(* Schneider Machine Expert - Basic project Modelo final v0.4, file version 2.6.0.0 *)
(* ProjectInformations: Name=Nuevo proyecto *)

HARDWARE
  Cpu 0: TM221CE24T
  EthernetConfiguration: NetworkName=M221, IpAllocationMode=FixedAddress, IpAddress=0.0.0.0, SubnetMask=0.0.0.0
  SerialLineConfiguration: Baud=Baud19200, Parity=ParityEven, DataBits=DataBits8, StopBits=StopBits1, PhysicalMedium=PhysicalMediumRs485, TransmissionMode=TransmissionModeModbusRtu, SlaveId=1, Addressing=SlaveAddressing
  MastTask: UsePeriodScanMode=false, PeriodScan=100
  FastTask: Period=255
  CpuBehavior: StartingMode=StartAsPreviousState, AutoSaveRamOnEeprom=true, WatchdogPeriod=250

SYMBOLS  (address, symbol, comment, settings)
  %M0         "Escalon frontal izquierdo"
  %M1         "Escalon frontal derecho"
  %M2         "Escalon trasero izquierdo"
  %M3         "Escalon trasero derecho"
  %M4         "Sensor frente izquierdo"
  %M5         "Sensor frente medio"
  %M6         "Sensor frente derecho"
  %M7         "Sensor derecha adelante"
  %M8         "Sensor derecha medio"
  %M9         "Sensor derecha atras"
  %M10        "Sensor trasero derecha"
  %M11        "Sensor trasero medio"
  %M12        "Sensor trasero izquierda"
  %M13        "Sensor izquierda atras"
  %M14        "Sensor izquierda medio"
  %M15        "Sensor izquierda adelante"
  %M16      FIFO_IN  "Carga en fifo"
  %M17      FIFO_OUT  "Descarga de fifo"
  %M20      FLAG1  "Cambio ΔNL o ΔNR"
  %M21      FLAG2  "Incrementos en Real"
  %M22      FLAG3  "Incrementos calculados"
  %M40      RST_S  "Reset/Enable Generador S"
  %M41      RST_DEMUX  "Reset/Enbale Demux"
  %M42      EN_ENCOD  "Enable Encoders"
  %M43      RST_ENCOD  "Reset Encoders"
  %M44      RST_FIFO  "Reset FIFOS"
  %M45      RST_STOP
  %M46      CONT_INIT  "Inicia contadores"
  %M47      CALC_CONST  "Calculo cte Cm"
  %M50      STP_MOV  "Stop Movement"
  %M51        "Enable Forward"
  %M52        "Enable Giro Horario"
  %M53        "Enable Giro A-Horario"
  %M54        "Enable F-G-H"
  %M55        "Enable F-G-AH"
  %M56        "Enable B-G-H"
  %M57        "Enable B-G-AH"
  %S6       SB_TB1S  "Base de tiempo de 1 s generada por un reloj interno"
  %MW10       "Buffer Distancia (WORD)"
  %MW11       "Buffer Velocidad"
  %MW12       "Buffer de Ratio/Angulo"
  %MW13       "Velocidad Izquierda"
  %MW14       "Velocidad Derecha"
  %MD0      PULSOS_L  "Diferencia %HSC0 - Preajuste"
  %MD2      PULSOS_R  "Diferencia %HSC1 - Preajuste"
  %MD4      PULSOS_L_ANTERIOR  "Num de cuenta intervalo anterior"
  %MD6      PULSOS_R_ANTERIOR  "Num de cuenta intervalo anterior"
  %MD8      ΔNL  "Delta pulsos encoder izq"
  %MD10     ΔNR  "Delta pulsos encoder der"
  %MF0      X_I  "X actual"
  %MF2      Y_I  "Y actual"
  %MF4      Θ_I  "θ actual"
  %MF6        "X Referencia"
  %MF8        "Y Referencia"
  %MF10       "θ Referencia"
  %MF12       "Xa - Xr"
  %MF14       "Ya - Yr"
  %MF16       "Distancia a la referencia"
  %MF18       "Modulo del buffer de distancia"
  %MF20       "Buffer de distancia (FLOAT)"
  %MF22     CM
  %MF24     ΔSL  "Delta movimiento lineal rueda izq"
  %MF26     ΔSR  "Delta movimiento lineal rueda der"
  %MF28     ΔSC  "Delta movimiento lineal mitad del eje"
  %MF30     ΔΘ  "Delta angular"
  %MF32     Θ_ANTERIOR  "Coordenada Θ intervalo anterior"
  %MF34     X_ANTERIOR  "Coordenada X intervalo anterior"
  %MF36     Y_ANTERIOR  "Coordenada Y intervalo anterior"
  %MF38     ΔNL_REAL  "Delta pulsos encoder izq en real"
  %MF40     ΔNR_REAL
  %KF0      PASOS  [Value=360]
  %KF2      RED  [Value=1]
  %KF4      PI  [Value=3.141592]
  %KF6      RADIO  [Value=0.083]
  %KF8      EJE  [Value=0.5]
  %TM0        [Preset=5, Base=OneHundredMilliSeconds]
  %TM1        [Preset=5, Base=OneHundredMilliSeconds]
  %TM2        [Preset=5, Base=OneHundredMilliSeconds]
  %TM3        [Preset=5, Base=OneHundredMilliSeconds]
  %TM4        [Preset=5, Base=OneHundredMilliSeconds]
  %TM5        [Preset=5, Base=OneHundredMilliSeconds]
  %TM6        [Preset=5, Base=OneHundredMilliSeconds]
  %TM7        [Preset=5, Base=OneHundredMilliSeconds]
  %TM8        [Preset=5, Base=OneHundredMilliSeconds]
  %TM9        [Preset=5, Base=OneHundredMilliSeconds]
  %TM10       [Preset=5, Base=OneHundredMilliSeconds]
  %TM11       [Preset=5, Base=OneHundredMilliSeconds]
  %TM12       [Preset=5, Base=OneHundredMilliSeconds]
  %TM13       [Preset=5, Base=OneHundredMilliSeconds]
  %TM14       [Preset=5, Base=OneHundredMilliSeconds]
  %TM15       [Preset=5, Base=OneHundredMilliSeconds]
  %C0         [Preset=17]
  %R0         "Distancia"
  %R1         "Velocidad"
  %R2         "Ratio Ruedas"
  %I0.0     ENC1A  "Encoder 1 A"
  %I0.1     ENC1B  "Encoder 1 B"
  %I0.6     ENC2A  "Encoder 2 A"
  %I0.7     ENC2B  "Encoder 2 B"
  %I0.8     MUX_IN  "Data de mux sensores"
  %Q0.0     L_PWM  "Salida PWM Motor Izquierdo"
  %Q0.1     R_PWM  "Salida PWM Motor Derecho"
  %Q0.2     L_DIR  "Salida Direccion Motor Izquierdo - 0:F 1:B"
  %Q0.3     R_DIR  "Salida Direccion Motor Derecho - 0:F 1:B"
  %Q0.4     S0  "MUX S0"
  %Q0.5     S1  "MUX S1"
  %Q0.6     S2  "MUX S2"
  %Q0.7     S3  "MUX S3"
  %Q0.8     LAMP0  "LAMPARAS BIT 0"
  %Q0.9     LAMP1  "LAMPARAS BIT 1"
  %HSC0       "Encoder Rueda Izquierda"  [Type=CounterOrDownCounterBiPhasesX2, Preset=2147483647, UseDoubleWord=true, DedicatedInputs(DedicatedInput(Activated=true), DedicatedInput(Activated=true)), ReflexOutputs(ReflexOutput(Activated=false, LessThanS0=false, GreaterOrEqualThanS0=false, GreaterOrEqualThanS1=false), ReflexOutput(Activated=false, LessThanS0=false, GreaterOrEqualThanS0=false, GreaterOrEqualThanS1=false)), Thresholds(Thresho]
  %HSC1       "Encoder Rueda Derecha"  [Type=CounterOrDownCounterBiPhasesX2, Preset=2147483647, UseDoubleWord=true, DedicatedInputs(DedicatedInput(Activated=true), DedicatedInput(Activated=true)), ReflexOutputs(ReflexOutput(Activated=false, LessThanS0=false, GreaterOrEqualThanS0=false, GreaterOrEqualThanS1=false), ReflexOutput(Activated=false, LessThanS0=false, GreaterOrEqualThanS0=false, GreaterOrEqualThanS1=false)), Thresholds(Thresho]
  %PWM0       "PWM_L"  [PtoObject(RefInput=NotUsed, ZPhaseInput=NotUsed, ProbeInput=NotUsed), GlobalIndex=0, Type=PWM, TimeBase=OneMilliSeconds, Preset=1]
  %PWM1       "PWM_R"  [PtoObject(RefInput=NotUsed, ZPhaseInput=NotUsed, ProbeInput=NotUsed), GlobalIndex=1, Type=PWM, TimeBase=OneMilliSeconds, Preset=1]

POU Demux
  (* SectionNumber=1 *)

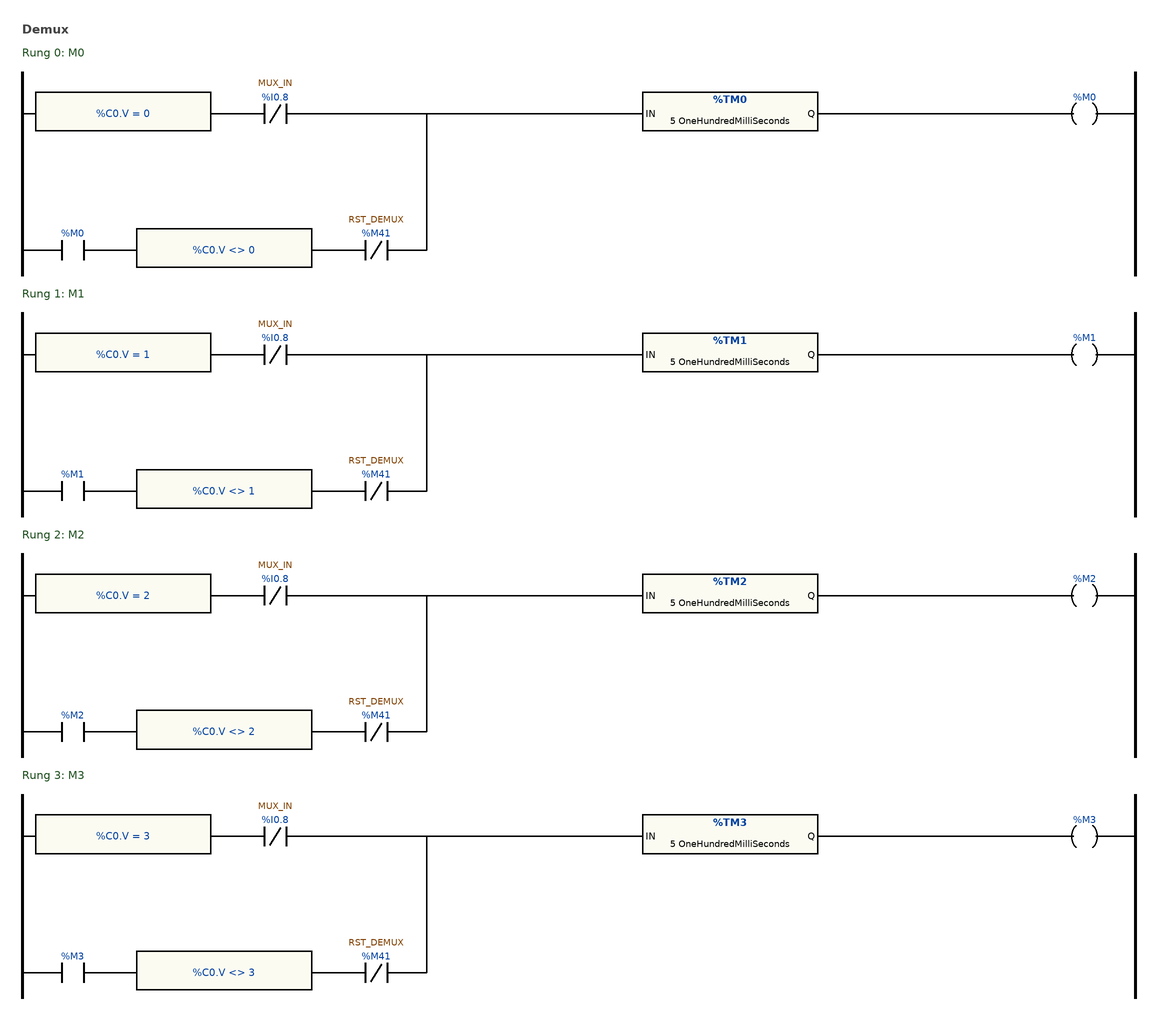

// Rung 0: M0
  BLK %TM0
  LD [ %C0.V = 0 ]
  ANDN %I0.8              (* MUX_IN *)
  OR( %M0
  AND [ %C0.V <> 0 ]
  ANDN %M41               (* RST_DEMUX *)
  )
  IN
  OUT_BLK
  LD Q
  ST %M0
  END_BLK
  // as ST:
  //   %TM0(IN := %C0.V = 0 AND NOT MUX_IN OR %M0 AND %C0.V <> 0 AND NOT RST_DEMUX);
  //   %M0 := %TM0.Q;

// Rung 1: M1
  BLK %TM1
  LD [ %C0.V = 1 ]
  ANDN %I0.8              (* MUX_IN *)
  OR( %M1
  AND [ %C0.V <> 1 ]
  ANDN %M41               (* RST_DEMUX *)
  )
  IN
  OUT_BLK
  LD Q
  ST %M1
  END_BLK
  // as ST:
  //   %TM1(IN := %C0.V = 1 AND NOT MUX_IN OR %M1 AND %C0.V <> 1 AND NOT RST_DEMUX);
  //   %M1 := %TM1.Q;

// Rung 2: M2
  BLK %TM2
  LD [ %C0.V = 2 ]
  ANDN %I0.8              (* MUX_IN *)
  OR( %M2
  AND [ %C0.V <> 2 ]
  ANDN %M41               (* RST_DEMUX *)
  )
  IN
  OUT_BLK
  LD Q
  ST %M2
  END_BLK
  // as ST:
  //   %TM2(IN := %C0.V = 2 AND NOT MUX_IN OR %M2 AND %C0.V <> 2 AND NOT RST_DEMUX);
  //   %M2 := %TM2.Q;

// Rung 3: M3
  BLK %TM3
  LD [ %C0.V = 3 ]
  ANDN %I0.8              (* MUX_IN *)
  OR( %M3
  AND [ %C0.V <> 3 ]
  ANDN %M41               (* RST_DEMUX *)
  )
  IN
  OUT_BLK
  LD Q
  ST %M3
  END_BLK
  // as ST:
  //   %TM3(IN := %C0.V = 3 AND NOT MUX_IN OR %M3 AND %C0.V <> 3 AND NOT RST_DEMUX);
  //   %M3 := %TM3.Q;

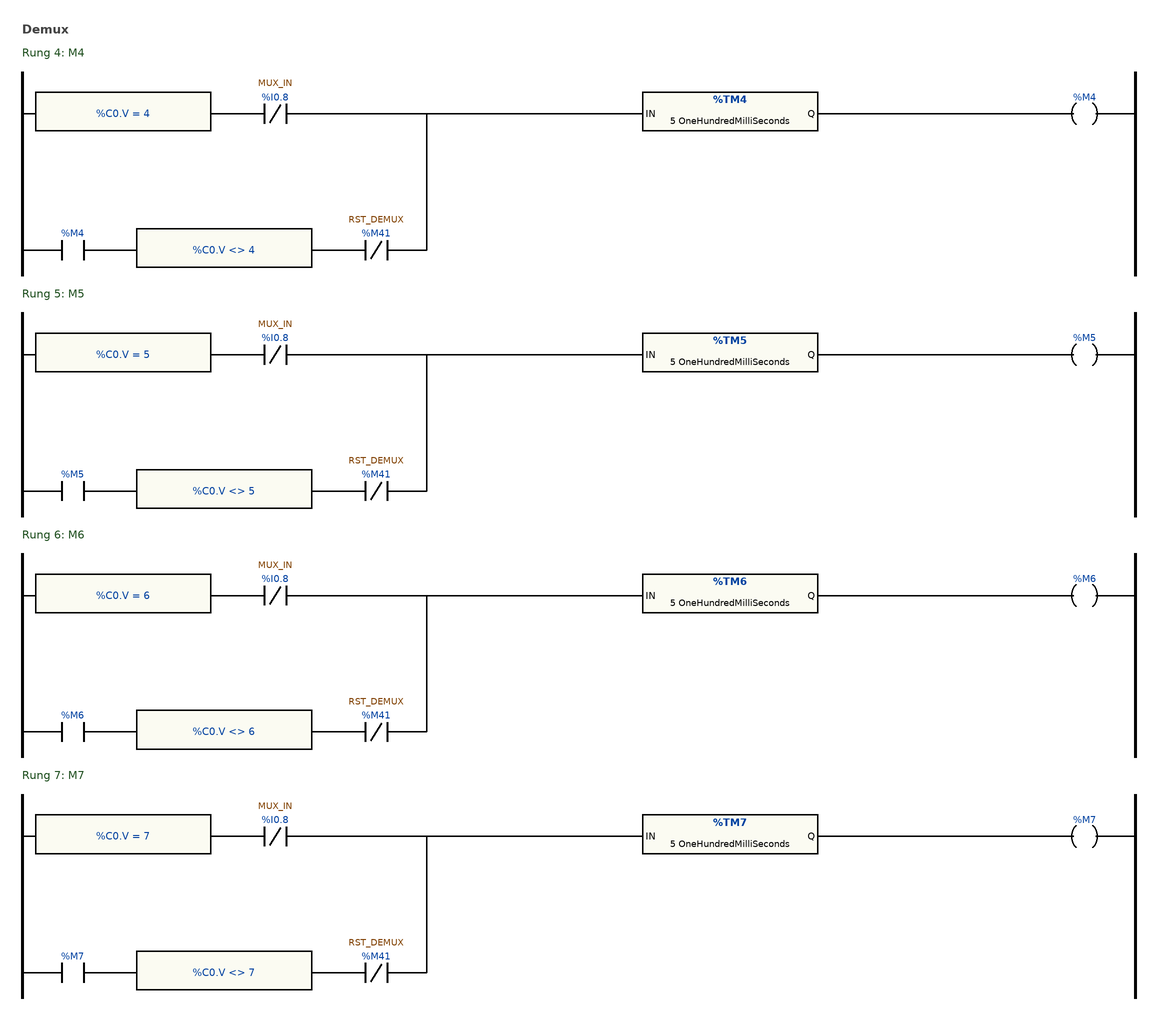

// Rung 4: M4
  BLK %TM4
  LD [ %C0.V = 4 ]
  ANDN %I0.8              (* MUX_IN *)
  OR( %M4
  AND [ %C0.V <> 4 ]
  ANDN %M41               (* RST_DEMUX *)
  )
  IN
  OUT_BLK
  LD Q
  ST %M4
  END_BLK
  // as ST:
  //   %TM4(IN := %C0.V = 4 AND NOT MUX_IN OR %M4 AND %C0.V <> 4 AND NOT RST_DEMUX);
  //   %M4 := %TM4.Q;

// Rung 5: M5
  BLK %TM5
  LD [ %C0.V = 5 ]
  ANDN %I0.8              (* MUX_IN *)
  OR( %M5
  AND [ %C0.V <> 5 ]
  ANDN %M41               (* RST_DEMUX *)
  )
  IN
  OUT_BLK
  LD Q
  ST %M5
  END_BLK
  // as ST:
  //   %TM5(IN := %C0.V = 5 AND NOT MUX_IN OR %M5 AND %C0.V <> 5 AND NOT RST_DEMUX);
  //   %M5 := %TM5.Q;

// Rung 6: M6
  BLK %TM6
  LD [ %C0.V = 6 ]
  ANDN %I0.8              (* MUX_IN *)
  OR( %M6
  AND [ %C0.V <> 6 ]
  ANDN %M41               (* RST_DEMUX *)
  )
  IN
  OUT_BLK
  LD Q
  ST %M6
  END_BLK
  // as ST:
  //   %TM6(IN := %C0.V = 6 AND NOT MUX_IN OR %M6 AND %C0.V <> 6 AND NOT RST_DEMUX);
  //   %M6 := %TM6.Q;

// Rung 7: M7
  BLK %TM7
  LD [ %C0.V = 7 ]
  ANDN %I0.8              (* MUX_IN *)
  OR( %M7
  AND [ %C0.V <> 7 ]
  ANDN %M41               (* RST_DEMUX *)
  )
  IN
  OUT_BLK
  LD Q
  ST %M7
  END_BLK
  // as ST:
  //   %TM7(IN := %C0.V = 7 AND NOT MUX_IN OR %M7 AND %C0.V <> 7 AND NOT RST_DEMUX);
  //   %M7 := %TM7.Q;

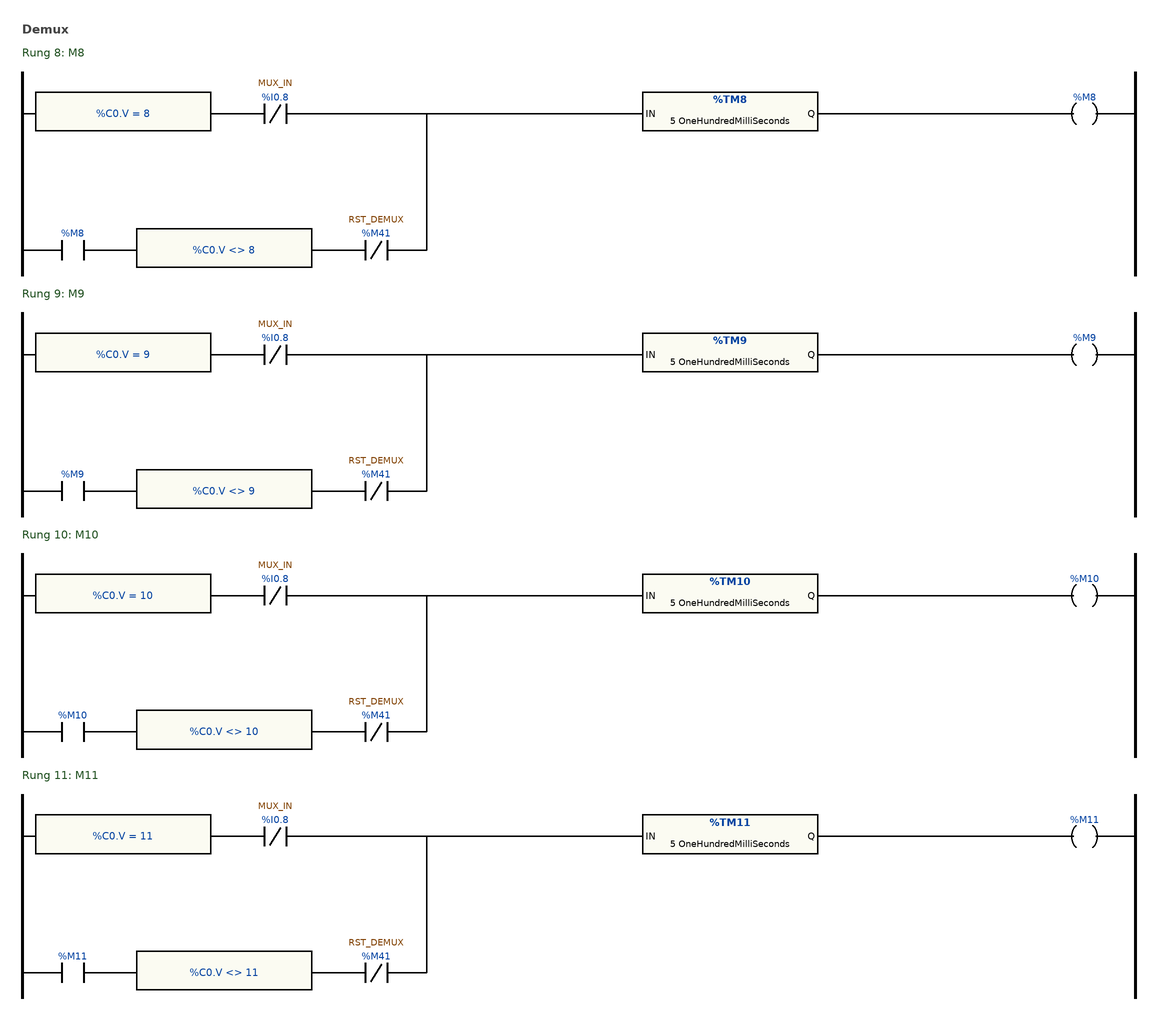

// Rung 8: M8
  BLK %TM8
  LD [ %C0.V = 8 ]
  ANDN %I0.8              (* MUX_IN *)
  OR( %M8
  AND [ %C0.V <> 8 ]
  ANDN %M41               (* RST_DEMUX *)
  )
  IN
  OUT_BLK
  LD Q
  ST %M8
  END_BLK
  // as ST:
  //   %TM8(IN := %C0.V = 8 AND NOT MUX_IN OR %M8 AND %C0.V <> 8 AND NOT RST_DEMUX);
  //   %M8 := %TM8.Q;

// Rung 9: M9
  BLK %TM9
  LD [ %C0.V = 9 ]
  ANDN %I0.8              (* MUX_IN *)
  OR( %M9
  AND [ %C0.V <> 9 ]
  ANDN %M41               (* RST_DEMUX *)
  )
  IN
  OUT_BLK
  LD Q
  ST %M9
  END_BLK
  // as ST:
  //   %TM9(IN := %C0.V = 9 AND NOT MUX_IN OR %M9 AND %C0.V <> 9 AND NOT RST_DEMUX);
  //   %M9 := %TM9.Q;

// Rung 10: M10
  BLK %TM10
  LD [ %C0.V = 10 ]
  ANDN %I0.8              (* MUX_IN *)
  OR( %M10
  AND [ %C0.V <> 10 ]
  ANDN %M41               (* RST_DEMUX *)
  )
  IN
  OUT_BLK
  LD Q
  ST %M10
  END_BLK
  // as ST:
  //   %TM10(IN := %C0.V = 10 AND NOT MUX_IN OR %M10 AND %C0.V <> 10 AND NOT RST_DEMUX);
  //   %M10 := %TM10.Q;

// Rung 11: M11
  BLK %TM11
  LD [ %C0.V = 11 ]
  ANDN %I0.8              (* MUX_IN *)
  OR( %M11
  AND [ %C0.V <> 11 ]
  ANDN %M41               (* RST_DEMUX *)
  )
  IN
  OUT_BLK
  LD Q
  ST %M11
  END_BLK
  // as ST:
  //   %TM11(IN := %C0.V = 11 AND NOT MUX_IN OR %M11 AND %C0.V <> 11 AND NOT RST_DEMUX);
  //   %M11 := %TM11.Q;

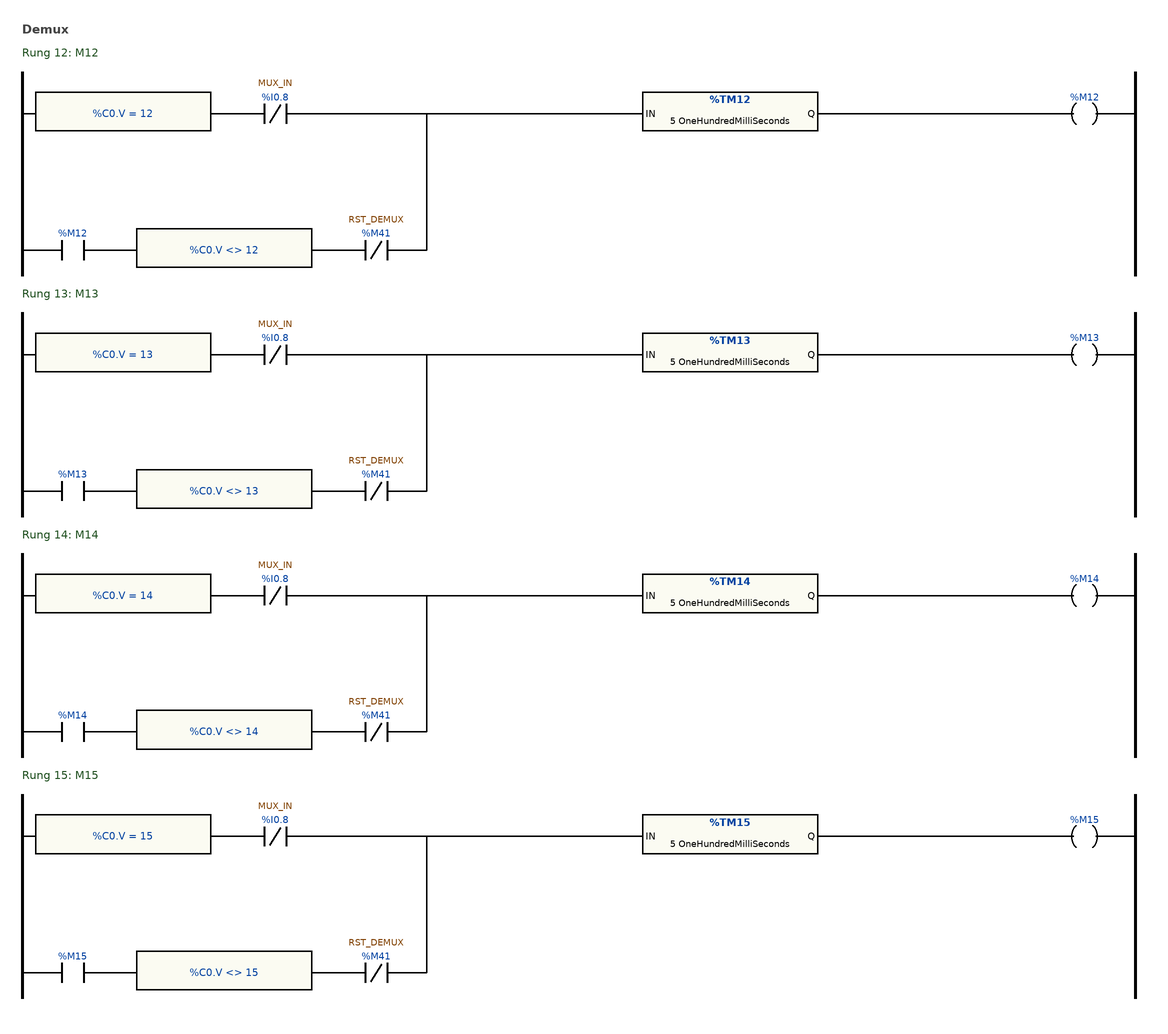

// Rung 12: M12
  BLK %TM12
  LD [ %C0.V = 12 ]
  ANDN %I0.8              (* MUX_IN *)
  OR( %M12
  AND [ %C0.V <> 12 ]
  ANDN %M41               (* RST_DEMUX *)
  )
  IN
  OUT_BLK
  LD Q
  ST %M12
  END_BLK
  // as ST:
  //   %TM12(IN := %C0.V = 12 AND NOT MUX_IN OR %M12 AND %C0.V <> 12 AND NOT RST_DEMUX);
  //   %M12 := %TM12.Q;

// Rung 13: M13
  BLK %TM13
  LD [ %C0.V = 13 ]
  ANDN %I0.8              (* MUX_IN *)
  OR( %M13
  AND [ %C0.V <> 13 ]
  ANDN %M41               (* RST_DEMUX *)
  )
  IN
  OUT_BLK
  LD Q
  ST %M13
  END_BLK
  // as ST:
  //   %TM13(IN := %C0.V = 13 AND NOT MUX_IN OR %M13 AND %C0.V <> 13 AND NOT RST_DEMUX);
  //   %M13 := %TM13.Q;

// Rung 14: M14
  BLK %TM14
  LD [ %C0.V = 14 ]
  ANDN %I0.8              (* MUX_IN *)
  OR( %M14
  AND [ %C0.V <> 14 ]
  ANDN %M41               (* RST_DEMUX *)
  )
  IN
  OUT_BLK
  LD Q
  ST %M14
  END_BLK
  // as ST:
  //   %TM14(IN := %C0.V = 14 AND NOT MUX_IN OR %M14 AND %C0.V <> 14 AND NOT RST_DEMUX);
  //   %M14 := %TM14.Q;

// Rung 15: M15
  BLK %TM15
  LD [ %C0.V = 15 ]
  ANDN %I0.8              (* MUX_IN *)
  OR( %M15
  AND [ %C0.V <> 15 ]
  ANDN %M41               (* RST_DEMUX *)
  )
  IN
  OUT_BLK
  LD Q
  ST %M15
  END_BLK
  // as ST:
  //   %TM15(IN := %C0.V = 15 AND NOT MUX_IN OR %M15 AND %C0.V <> 15 AND NOT RST_DEMUX);
  //   %M15 := %TM15.Q;

POU Generacion Sx
  (* SectionNumber=2 *)

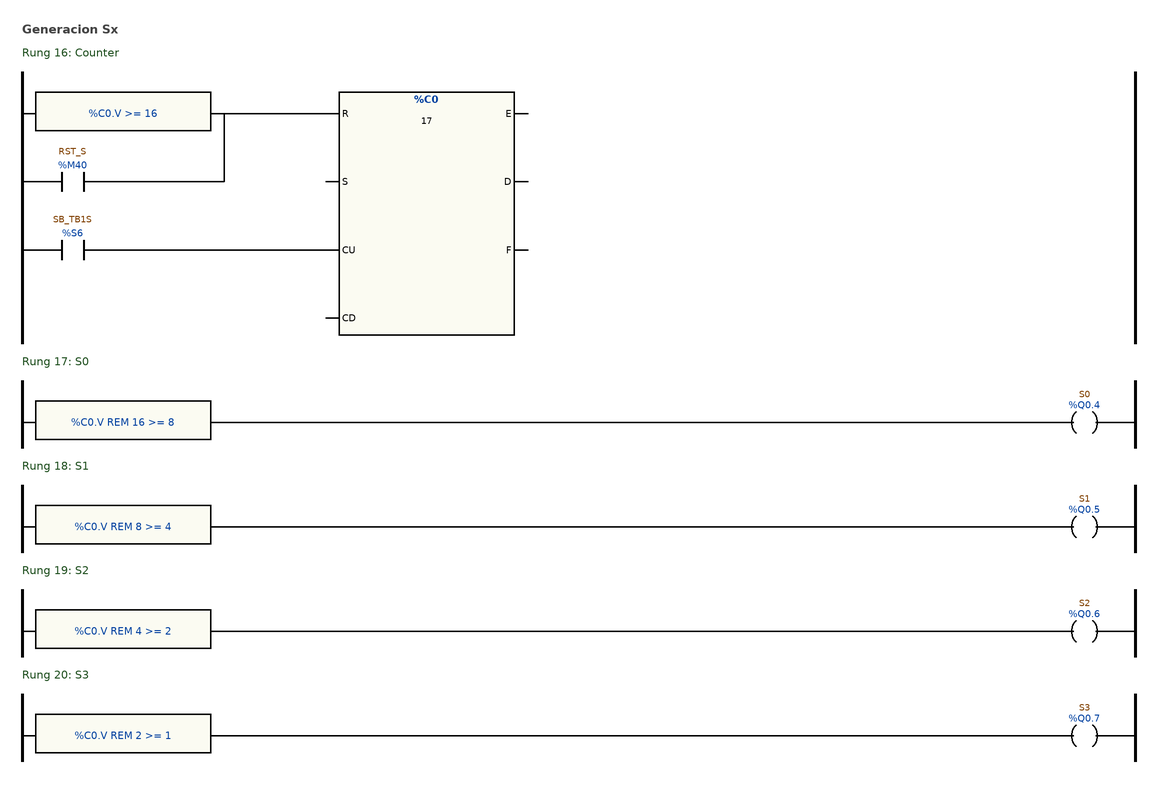

// Rung 16: Counter
  BLK %C0
  LD [ %C0.V >= 16 ]
  OR %M40                 (* RST_S *)
  R
  LD %S6                  (* SB_TB1S *)
  CU
  END_BLK
  // as ST:
  //   %C0(R := %C0.V >= 16 OR RST_S, CU := SB_TB1S);

// Rung 17: S0
  LD 1
  AND [%C0.V REM 16 >= 8]
  ST %Q0.4                (* S0 *)
  // as ST:
  //   S0 := %C0.V REM 16 >= 8;

// Rung 18: S1
  LD 1
  AND [%C0.V REM 8 >= 4]
  ST %Q0.5                (* S1 *)
  // as ST:
  //   S1 := %C0.V REM 8 >= 4;

// Rung 19: S2
  LD 1
  AND [%C0.V REM 4 >= 2]
  ST %Q0.6                (* S2 *)
  // as ST:
  //   S2 := %C0.V REM 4 >= 2;

// Rung 20: S3
  LD 1
  AND [%C0.V REM 2 >= 1]
  ST %Q0.7                (* S3 *)
  // as ST:
  //   S3 := %C0.V REM 2 >= 1;

POU Control de Motores
  (* SectionNumber=3 *)

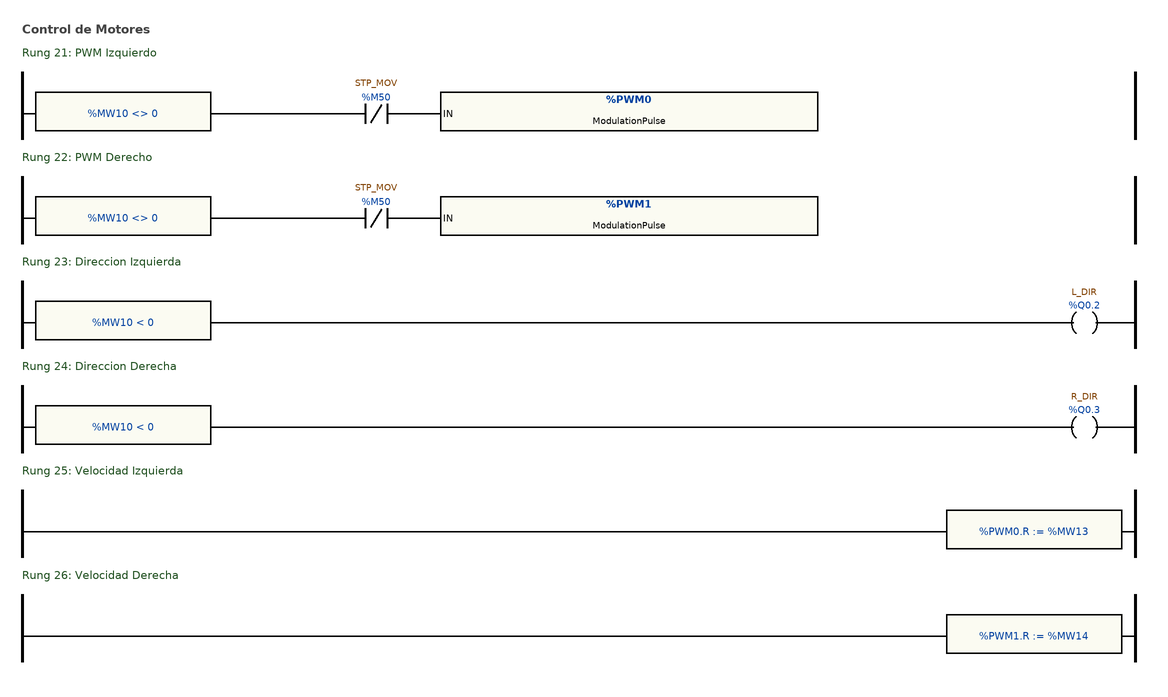

// Rung 21: PWM Izquierdo
  BLK %PWM0
  LD [ %MW10 <> 0 ]
  ANDN %M50               (* STP_MOV *)
  IN
  END_BLK
  // as ST:
  //   %PWM0(IN := %MW10 <> 0 AND NOT STP_MOV);

// Rung 22: PWM Derecho
  BLK %PWM1
  LD [ %MW10 <> 0 ]
  ANDN %M50               (* STP_MOV *)
  IN
  END_BLK
  // as ST:
  //   %PWM1(IN := %MW10 <> 0 AND NOT STP_MOV);

// Rung 23: Direccion Izquierda
  LD [ %MW10 < 0 ]
  ST %Q0.2                (* L_DIR *)
  // as ST:
  //   L_DIR := %MW10 < 0;

// Rung 24: Direccion Derecha
  LD [ %MW10 < 0 ]
  ST %Q0.3                (* R_DIR *)
  // as ST:
  //   R_DIR := %MW10 < 0;

// Rung 25: Velocidad Izquierda
  LD 1
  [ %PWM0.R := %MW13 ]
  // as ST:
  //   %PWM0.R := %MW13;

// Rung 26: Velocidad Derecha
  LD 1
  [ %PWM1.R := %MW14 ]
  // as ST:
  //   %PWM1.R := %MW14;

POU FIFOS
  (* SectionNumber=4 *)

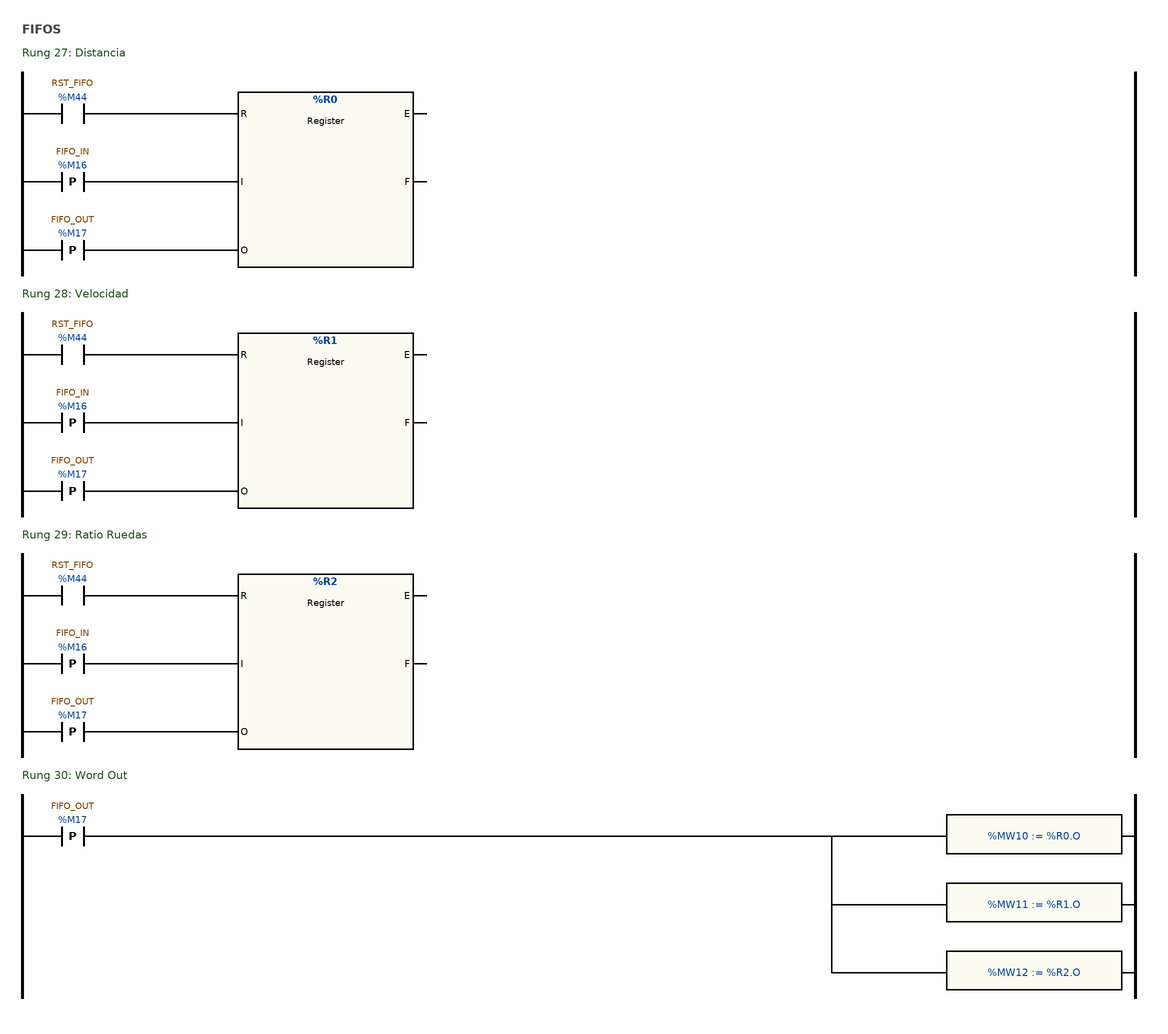

// Rung 27: Distancia
  BLK %R0
  LD %M44                 (* RST_FIFO *)
  R
  LDR %M16                (* FIFO_IN *)
  I
  LDR %M17                (* FIFO_OUT *)
  O
  END_BLK
  // as ST:
  //   %R0(R := RST_FIFO, I := RISING(FIFO_IN), O := RISING(FIFO_OUT));

// Rung 28: Velocidad
  BLK %R1
  LD %M44                 (* RST_FIFO *)
  R
  LDR %M16                (* FIFO_IN *)
  I
  LDR %M17                (* FIFO_OUT *)
  O
  END_BLK
  // as ST:
  //   %R1(R := RST_FIFO, I := RISING(FIFO_IN), O := RISING(FIFO_OUT));

// Rung 29: Ratio Ruedas
  BLK %R2
  LD %M44                 (* RST_FIFO *)
  R
  LDR %M16                (* FIFO_IN *)
  I
  LDR %M17                (* FIFO_OUT *)
  O
  END_BLK
  // as ST:
  //   %R2(R := RST_FIFO, I := RISING(FIFO_IN), O := RISING(FIFO_OUT));

// Rung 30: Word Out
  LDR %M17                (* FIFO_OUT *)
  [ %MW10 := %R0.O ]
  [ %MW11 := %R1.O ]
  [ %MW12 := %R2.O ]
  // as ST:
  //   IF RISING(FIFO_OUT) THEN %MW10 := %R0.O; END_IF;
  //   IF RISING(FIFO_OUT) THEN %MW11 := %R1.O; END_IF;
  //   IF RISING(FIFO_OUT) THEN %MW12 := %R2.O; END_IF;

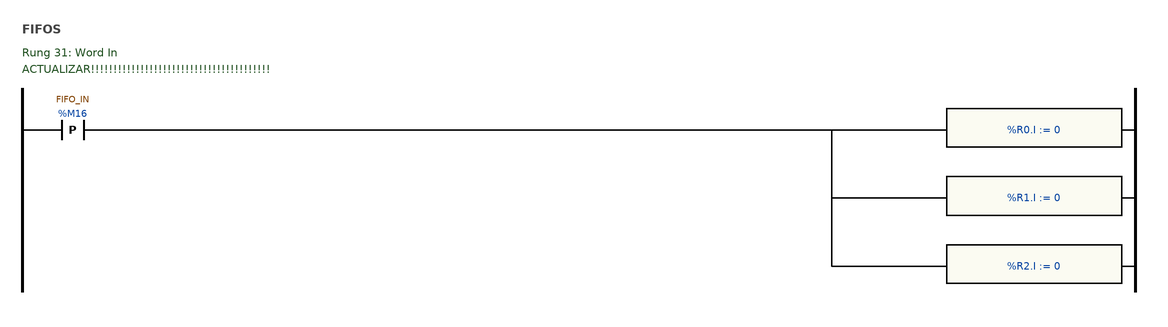

// Rung 31: Word In
// ACTUALIZAR!!!!!!!!!!!!!!!!!!!!!!!!!!!!!!!!!!!!!!!!
  LDR %M16                (* FIFO_IN *)
  [ %R0.I := 0 ]
  [ %R1.I := 0 ]
  [ %R2.I := 0 ]
  // as ST:
  //   IF RISING(FIFO_IN) THEN %R0.I := 0; END_IF;
  //   IF RISING(FIFO_IN) THEN %R1.I := 0; END_IF;
  //   IF RISING(FIFO_IN) THEN %R2.I := 0; END_IF;

POU Control de Colision
  (* SectionNumber=5 *)

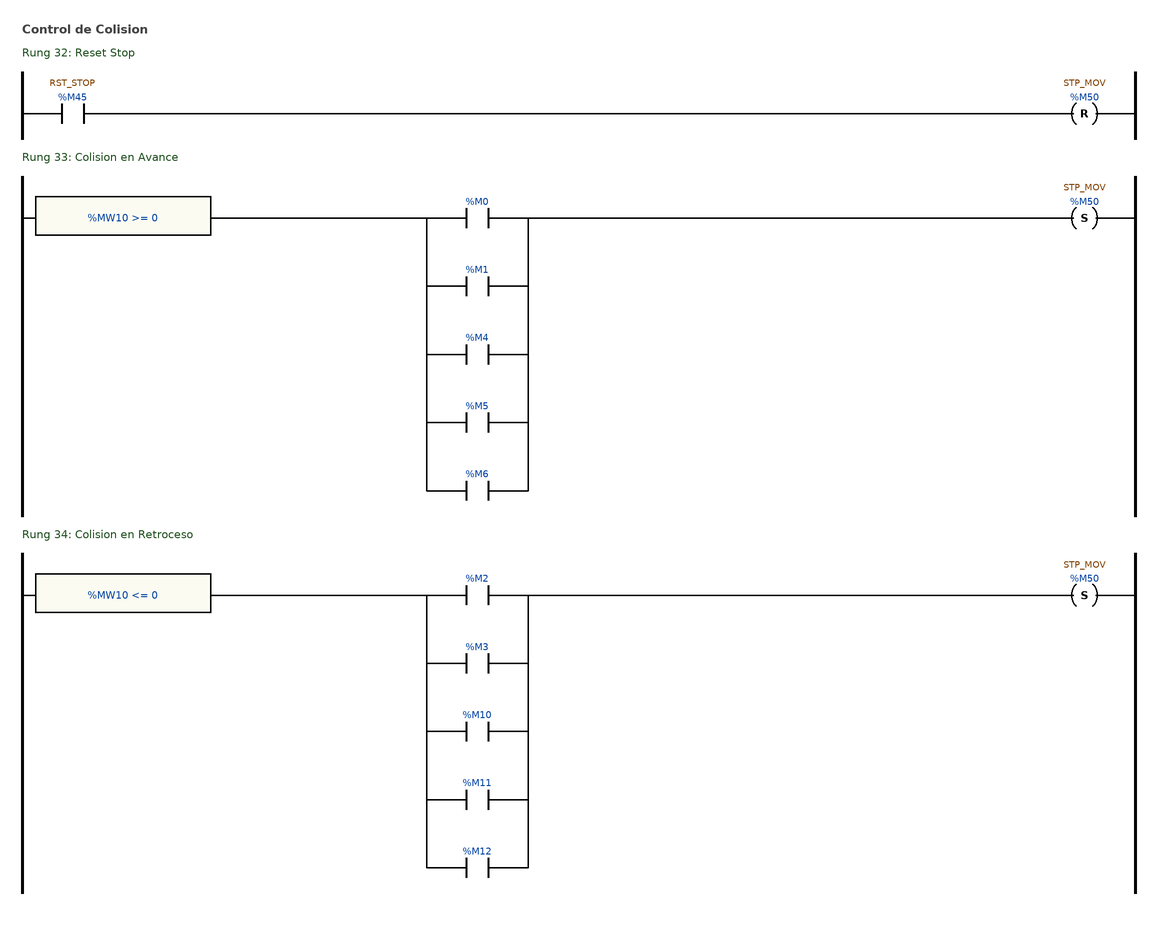

// Rung 32: Reset Stop
  LD %M45                 (* RST_STOP *)
  R %M50                  (* STP_MOV *)
  // as ST:
  //   IF RST_STOP THEN STP_MOV := FALSE; END_IF;

// Rung 33: Colision en Avance
  LD [ %MW10 >= 0 ]
  AND( %M0
  OR %M1
  OR %M4
  OR %M5
  OR %M6
  )
  S %M50                  (* STP_MOV *)
  // as ST:
  //   IF %MW10 >= 0 AND (%M0 OR %M1 OR %M4 OR %M5 OR %M6) THEN STP_MOV := TRUE; END_IF;

// Rung 34: Colision en Retroceso
  LD [ %MW10 <= 0 ]
  AND( %M2
  OR %M3
  OR %M10
  OR %M11
  OR %M12
  )
  S %M50                  (* STP_MOV *)
  // as ST:
  //   IF %MW10 <= 0 AND (%M2 OR %M3 OR %M10 OR %M11 OR %M12) THEN STP_MOV := TRUE; END_IF;

POU Traduccion de Comandos
  (* SectionNumber=6 *)

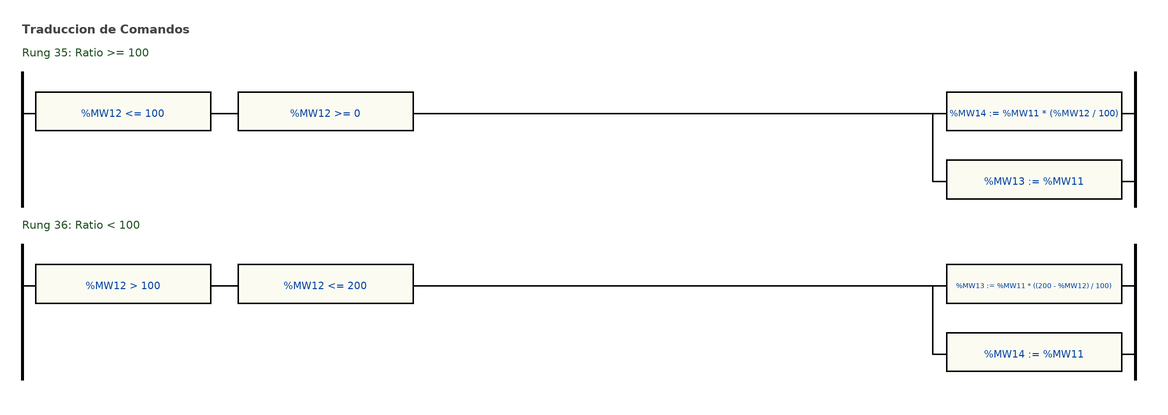

// Rung 35: Ratio >= 100
  LD [ %MW12 <= 100 ]
  AND [ %MW12 >= 0 ]
  [%MW14 := %MW11 * (%MW12 / 100)]
  [ %MW13 := %MW11 ]
  // as ST:
  //   IF %MW12 <= 100 AND %MW12 >= 0 THEN %MW14 := %MW11 * (%MW12 / 100); END_IF;
  //   IF %MW12 <= 100 AND %MW12 >= 0 THEN %MW13 := %MW11; END_IF;

// Rung 36: Ratio < 100
  LD [ %MW12 > 100 ]
  AND [ %MW12 <= 200 ]
  [%MW13 := %MW11 * ((200 - %MW12) / 100)]
  [ %MW14 := %MW11 ]
  // as ST:
  //   IF %MW12 > 100 AND %MW12 <= 200 THEN %MW13 := %MW11 * ((200 - %MW12) / 100); END_IF;
  //   IF %MW12 > 100 AND %MW12 <= 200 THEN %MW14 := %MW11; END_IF;

POU Realimentacion Distancia  (* Guarda la distancia cuando se hace una bajada del FIFO y calcula la distancia avanzada desde ese punto *)
  (* SectionNumber=7 *)

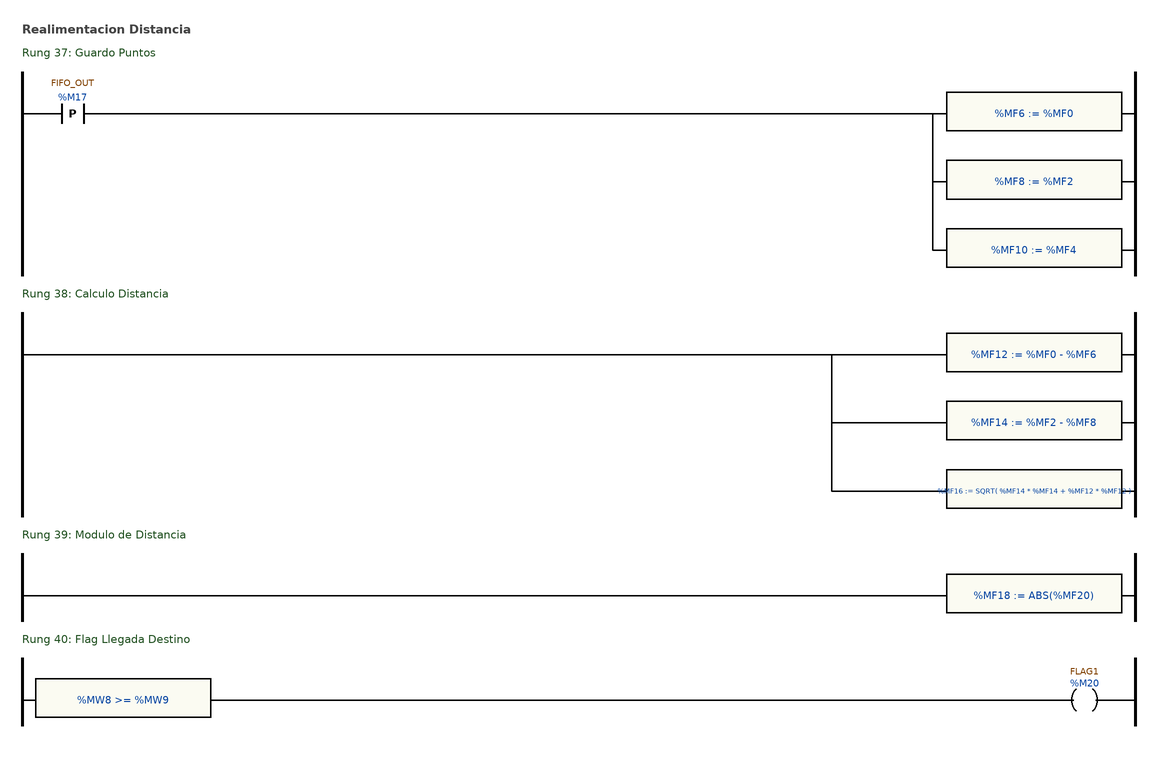

// Rung 37: Guardo Puntos
  LDR %M17                (* FIFO_OUT *)
  [ %MF6 := %MF0 ]        (* X_I *)
  [ %MF8 := %MF2 ]        (* Y_I *)
  [ %MF10 := %MF4 ]       (* Θ_I *)
  // as ST:
  //   IF RISING(FIFO_OUT) THEN %MF6 := X_I; END_IF;
  //   IF RISING(FIFO_OUT) THEN %MF8 := Y_I; END_IF;
  //   IF RISING(FIFO_OUT) THEN %MF10 := Θ_I; END_IF;

// Rung 38: Calculo Distancia
  LD 1
  [ %MF12 := %MF0 - %MF6 ](* X_I *)
  [ %MF14 := %MF2 - %MF8 ](* Y_I *)
  [%MF16 := SQRT( %MF14 * %MF14 + %MF12 * %MF12 )]
  // as ST:
  //   %MF12 := X_I - %MF6;
  //   %MF14 := Y_I - %MF8;
  //   %MF16 := SQRT( %MF14 * %MF14 + %MF12 * %MF12 );

// Rung 39: Modulo de Distancia
  LD 1
  [ %MF18 := ABS ( %MF20 ) ]
  // as ST:
  //   %MF18 := ABS ( %MF20 );

// Rung 40: Flag Llegada Destino
  LD [ %MW8 >= %MW9 ]
  ST %M20                 (* FLAG1 *)
  // as ST:
  //   FLAG1 := %MW8 >= %MW9;

POU Contadores
  (* SectionNumber=8 *)

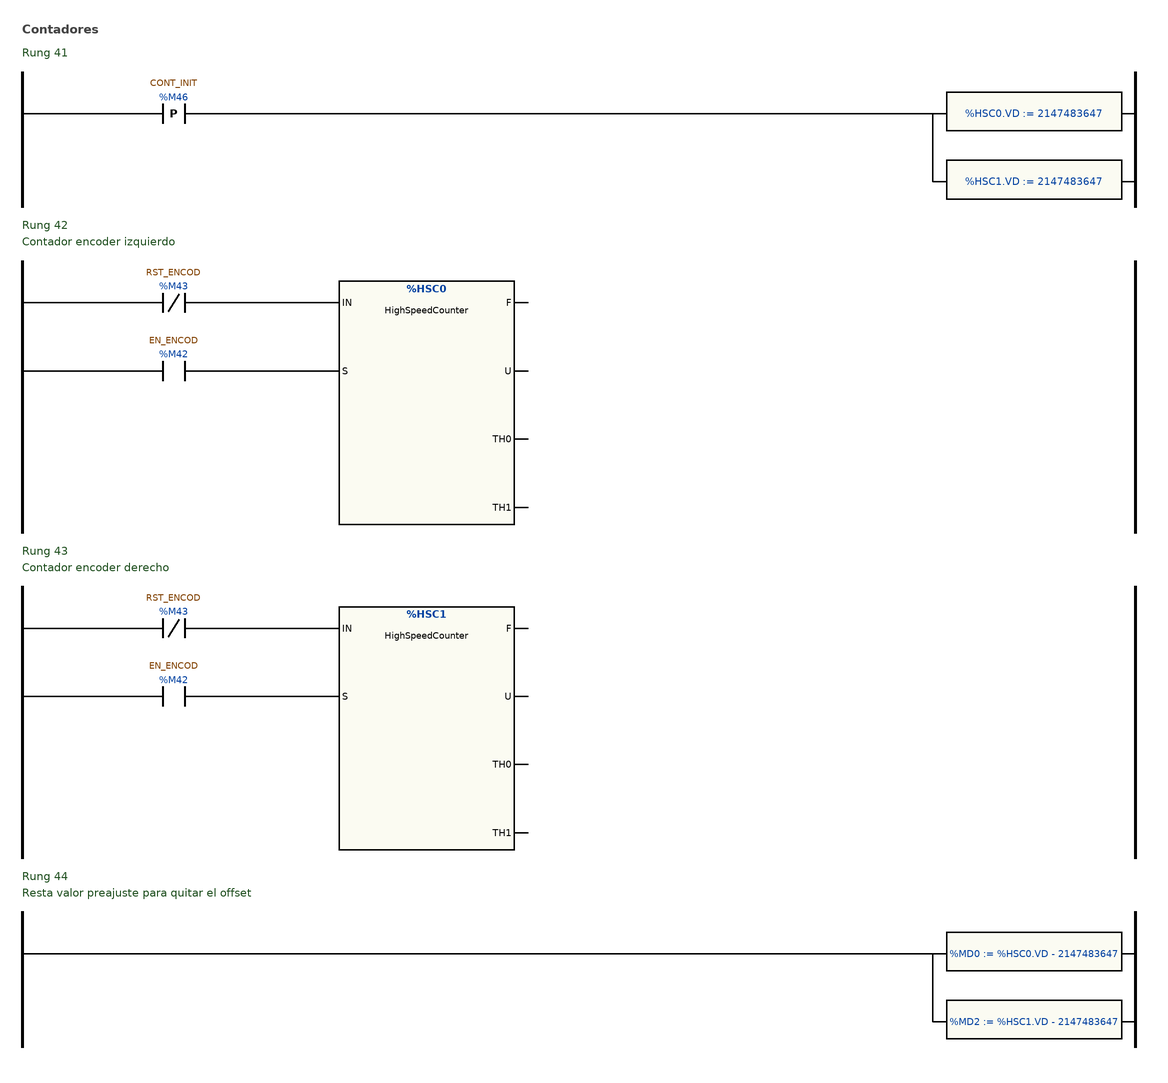

// Rung 41
  LDR %M46                (* CONT_INIT *)
  [ %HSC0.VD := 2147483647 ]
  [ %HSC1.VD := 2147483647 ]
  // as ST:
  //   IF RISING(CONT_INIT) THEN %HSC0.VD := 2147483647; END_IF;
  //   IF RISING(CONT_INIT) THEN %HSC1.VD := 2147483647; END_IF;

// Rung 42
// Contador encoder izquierdo
  BLK %HSC0
  LDN %M43                (* RST_ENCOD *)
  IN
  LD %M42                 (* EN_ENCOD *)
  S
  END_BLK
  // as ST:
  //   %HSC0(IN := NOT RST_ENCOD, S := EN_ENCOD);

// Rung 43
// Contador encoder derecho
  BLK %HSC1
  LDN %M43                (* RST_ENCOD *)
  IN
  LD %M42                 (* EN_ENCOD *)
  S
  END_BLK
  // as ST:
  //   %HSC1(IN := NOT RST_ENCOD, S := EN_ENCOD);

// Rung 44
// Resta valor preajuste para quitar el offset
  LD 1
  [ %MD0 := %HSC0.VD - 2147483647 ](* PULSOS_L *)
  [ %MD2 := %HSC1.VD - 2147483647 ](* PULSOS_R *)
  // as ST:
  //   PULSOS_L := %HSC0.VD - 2147483647;
  //   PULSOS_R := %HSC1.VD - 2147483647;

POU Constantes
  (* SectionNumber=9 *)

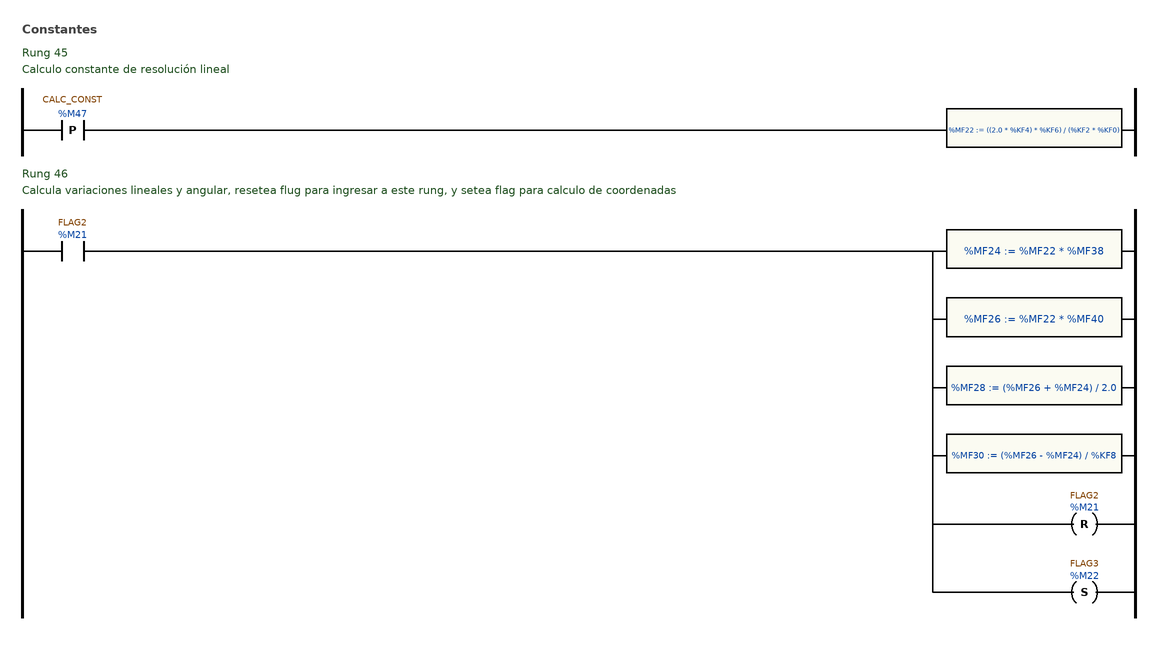

// Rung 45
// Calculo constante de resolución lineal
  LDR %M47                (* CALC_CONST *)
  [ %MF22 := ( ( 2.0 * %KF4 ) * %KF6 ) / ( %KF2 * %KF0 ) ](* CM, PI, RADIO, RED, PASOS *)
  // as ST:
  //   IF RISING(CALC_CONST) THEN CM := ( ( 2.0 * PI ) * RADIO ) / ( RED * PASOS ); END_IF;

// Rung 46
// Calcula variaciones lineales y angular, resetea flug para ingresar a este rung, y setea flag para calculo de coordenadas
  LD %M21                 (* FLAG2 *)
  [ %MF24 := %MF22 * %MF38 ](* ΔSL, CM, ΔNL_REAL *)
  [ %MF26 := %MF22 * %MF40 ](* ΔSR, CM, ΔNR_REAL *)
  [%MF28 := (%MF26 + %MF24) / 2.0](* ΔSC, ΔSR, ΔSL *)
  [%MF30 := (%MF26 - %MF24) / %KF8](* ΔΘ, ΔSR, ΔSL, EJE *)
  R %M21                  (* FLAG2 *)
  S %M22                  (* FLAG3 *)
  // as ST:
  //   IF FLAG2 THEN ΔSL := CM * ΔNL_REAL; END_IF;
  //   IF FLAG2 THEN ΔSR := CM * ΔNR_REAL; END_IF;
  //   IF FLAG2 THEN ΔSC := (ΔSR + ΔSL) / 2.0; END_IF;
  //   IF FLAG2 THEN ΔΘ := (ΔSR - ΔSL) / EJE; END_IF;
  //   _t1 := FLAG2;
  //   IF _t1 THEN FLAG2 := FALSE; END_IF;
  //   IF _t1 THEN FLAG3 := TRUE; END_IF;

POU Delta pulsos
  (* SectionNumber=10 *)

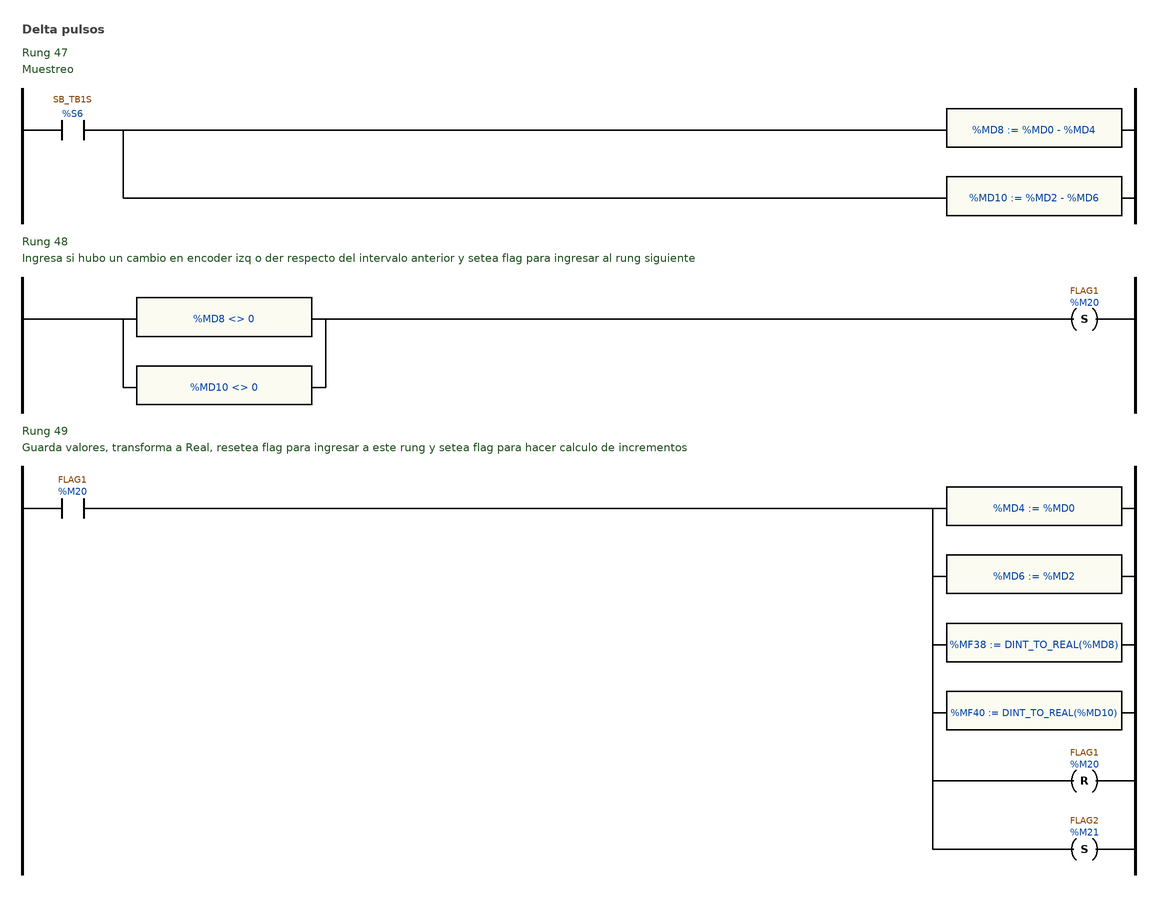

// Rung 47
// Muestreo
  LD %S6                  (* SB_TB1S *)
  [ %MD8 := %MD0 - %MD4 ] (* ΔNL, PULSOS_L, PULSOS_L_ANTERIOR *)
  [ %MD10 := %MD2 - %MD6 ](* ΔNR, PULSOS_R, PULSOS_R_ANTERIOR *)
  // as ST:
  //   IF SB_TB1S THEN ΔNL := PULSOS_L - PULSOS_L_ANTERIOR; END_IF;
  //   IF SB_TB1S THEN ΔNR := PULSOS_R - PULSOS_R_ANTERIOR; END_IF;

// Rung 48
// Ingresa si hubo un cambio en encoder izq o der respecto del intervalo anterior y setea flag para ingresar al rung siguiente
  LD 1
  AND( [ %MD8 <> 0 ]      (* ΔNL *)
  OR [ %MD10 <> 0 ]       (* ΔNR *)
  )
  S %M20                  (* FLAG1 *)
  // as ST:
  //   IF ΔNL <> 0 OR ΔNR <> 0 THEN FLAG1 := TRUE; END_IF;

// Rung 49
// Guarda valores, transforma a Real, resetea flag para ingresar a este rung y setea flag para hacer calculo de incrementos
  LD %M20                 (* FLAG1 *)
  [ %MD4 := %MD0 ]        (* PULSOS_L_ANTERIOR, PULSOS_L *)
  [ %MD6 := %MD2 ]        (* PULSOS_R_ANTERIOR, PULSOS_R *)
  [ %MF38 := DINT_TO_REAL ( %MD8 ) ](* ΔNL_REAL, ΔNL *)
  [ %MF40 := DINT_TO_REAL ( %MD10 ) ](* ΔNR_REAL, ΔNR *)
  R %M20                  (* FLAG1 *)
  S %M21                  (* FLAG2 *)
  // as ST:
  //   IF FLAG1 THEN PULSOS_L_ANTERIOR := PULSOS_L; END_IF;
  //   IF FLAG1 THEN PULSOS_R_ANTERIOR := PULSOS_R; END_IF;
  //   IF FLAG1 THEN ΔNL_REAL := DINT_TO_REAL ( ΔNL ); END_IF;
  //   IF FLAG1 THEN ΔNR_REAL := DINT_TO_REAL ( ΔNR ); END_IF;
  //   _t1 := FLAG1;
  //   IF _t1 THEN FLAG1 := FALSE; END_IF;
  //   IF _t1 THEN FLAG2 := TRUE; END_IF;

POU Calculo coordenadas
  (* SectionNumber=11 *)

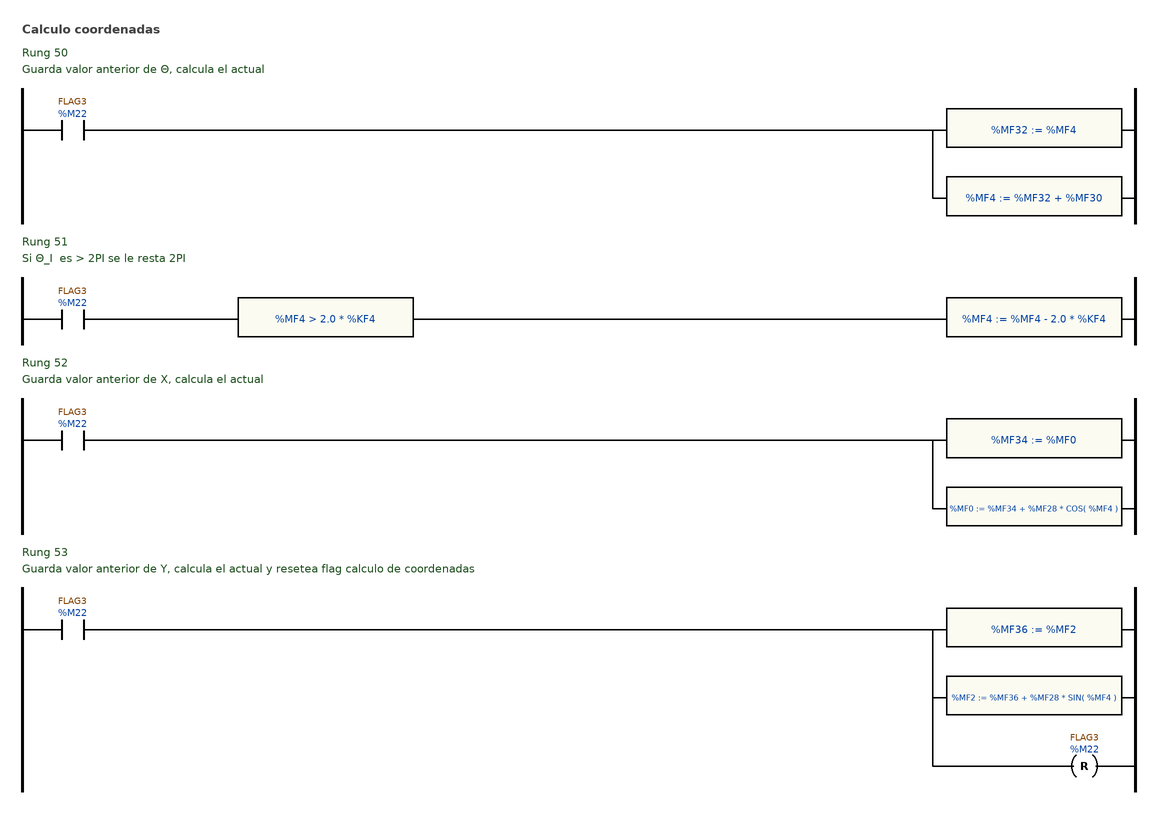

// Rung 50
// Guarda valor anterior de Θ, calcula el actual
  LD %M22                 (* FLAG3 *)
  [ %MF32 := %MF4 ]       (* Θ_ANTERIOR, Θ_I *)
  [ %MF4 := %MF32 + %MF30 ](* Θ_I, Θ_ANTERIOR, ΔΘ *)
  // as ST:
  //   IF FLAG3 THEN Θ_ANTERIOR := Θ_I; END_IF;
  //   IF FLAG3 THEN Θ_I := Θ_ANTERIOR + ΔΘ; END_IF;

// Rung 51
// Si Θ_I  es > 2PI se le resta 2PI
  LD %M22                 (* FLAG3 *)
  AND [%MF4 > 2.0 * %KF4] (* Θ_I, PI *)
  [%MF4 := %MF4 - 2.0 * %KF4](* Θ_I, Θ_I, PI *)
  // as ST:
  //   IF FLAG3 AND Θ_I > 2.0 * PI THEN Θ_I := Θ_I - 2.0 * PI; END_IF;

// Rung 52
// Guarda valor anterior de X, calcula el actual
  LD %M22                 (* FLAG3 *)
  [ %MF34 := %MF0 ]       (* X_ANTERIOR, X_I *)
  [%MF0 := %MF34 + %MF28 * COS( %MF4 )](* X_I, X_ANTERIOR, ΔSC, Θ_I *)
  // as ST:
  //   IF FLAG3 THEN X_ANTERIOR := X_I; END_IF;
  //   IF FLAG3 THEN X_I := X_ANTERIOR + ΔSC * COS( Θ_I ); END_IF;

// Rung 53
// Guarda valor anterior de Y, calcula el actual y resetea flag calculo de coordenadas
  LD %M22                 (* FLAG3 *)
  [ %MF36 := %MF2 ]       (* Y_ANTERIOR, Y_I *)
  [%MF2 := %MF36 + %MF28 * SIN( %MF4 )](* Y_I, Y_ANTERIOR, ΔSC, Θ_I *)
  R %M22                  (* FLAG3 *)
  // as ST:
  //   IF FLAG3 THEN Y_ANTERIOR := Y_I; END_IF;
  //   IF FLAG3 THEN Y_I := Y_ANTERIOR + ΔSC * SIN( Θ_I ); END_IF;
  //   IF FLAG3 THEN FLAG3 := FALSE; END_IF;
